{attribute 'strict'}
{attribute 'to_string'}
TYPE ENUM_STATION :
(
	SCREWING:= 0,
	GSL:= 1,
	DISPENSER:= 2
);
END_TYPE

(* stored: Version 1.1.0.1, ProductVersion 3.1.4024.10
   DUT ENUM_STATION: Id {ecbeddc3-2b1c-4d7f-a5d6-7e27d5901849} *)
